{attribute 'GeneratedUsingTerminal: EL3773-0000-0018'}
{attribute addProperty BoxType "EL3773-0000-0018"}
{attribute addProperty Id "U3_SamplesAT %I*U3_Samples_2D13B74B20"}
{attribute addProperty CRC "3050289389"}
{attribute addProperty Size "20"}
TYPE L3_Voltage_Samples_B5CFB8ED EXTENDS InputBase_8311D824 :
STRUCT
	{attribute addProperty Name "U3_Samples"}
	U3_Samples AT %I* : U3_Samples_2D13B74B;
END_STRUCT
END_TYPE

(* stored: Version 1.2.0.0, ProductVersion 3.1.4024.9
   DUT L3_Voltage_Samples_B5CFB8ED: Id {d7a6921d-3558-4822-9a5e-95058c2aef89} *)
